TYPE Patient :
STRUCT
	X : DINT := -10000; //patient location in mm
	Y : DINT := -10000; //patient location in mm
	ActiveSwitch: BOOL;
	AgeTimer : TON;
	AGE: TIME := T#0S;
END_STRUCT
END_TYPE

(* stored: Version 1.1.0.1, ProductVersion 3.1.4022.3
   DUT Patient: Id {7326ef91-ac2a-4ed4-9579-abaabf1bab05} *)
